	DATA_BLOCK DB163
	TITLE =DBG063M  AERATION AIR STEEPING 16
	//COPYRIGHT:    (C) 2009  BUHLER AG, CH-9240 UZWIL, SWITZERLAND
	//
	//PRODUCT:      WinCoS_BIW01_09
	//
	//TITLE:        AERATION AIR STEEPING 16
	//                Machine group DB
	//                Maschinengruppen-DB
	//
	//-------------------------------------------------------------------------
	//
	//IDENT:        AUTHOR:             DEPT:             DATE:
	//
	//P01_DB163.1.0 K.Renz              CSB41             13.Jan.2010
	//              1st Release
	//
	//-------------------------------------------------------------------------
	//
	//PURPOSE:
	//
	//MANUAL :
	//
	//RESTRICTIONS:
	//
	//-------------------------------------------------------------------------
	AUTHOR  : KR
	FAMILY  : USW
	NAME    : DBG063M
	VERSION : 00.00

	FB163
	BEGIN
	      #Gr.Par.ParObjectNo 	:=6300;
	      #Gr.Par.ParIdling      	:=2;
	      #Gr.Par.ParMgr	        :=True;
	      #Gr.Par.ParWgr	        :=False;
	      #Gr.Par.ParGgr	        :=False;
	      #Gr.Par.ParEmptyingTime 	:=0;
	      #Gr.Par.ParHornCode       :=1;
	//Parameter =A-1126-QXV/BZS41/42 : AERATION AIR RING ST 16
	      #A_1126_QXV_BZS41_42.Par.ParObjectNo                             :=6301;
	      #A_1126_QXV_BZS41_42.Par.ParMsgType                              :=7081;
	      #A_1126_QXV_BZS41_42.Par.ParHornCode                             :=1;
	      #A_1126_QXV_BZS41_42.Par.ParMonTime                              :=100;
	      #A_1126_QXV_BZS41_42.Par.ParPulseTimeHN                          :=5;
	      #A_1126_QXV_BZS41_42.Par.ParPulseTimeLN                          :=5;
	      #A_1126_QXV_BZS41_42.Par.ParIdlingTime                           :=0;
	      #A_1126_QXV_BZS41_42.Par.ParDelayTime                            :=0;
	      #A_1126_QXV_BZS41_42.Par.ParLogOff                               :=False;
	      #A_1126_QXV_BZS41_42.Par.ParManual                               :=True;
	      #A_1126_QXV_BZS41_42.Par.ParPulseValve                           :=False;
	      #A_1126_QXV_BZS41_42.Par.ParContValve                            :=True;
	      #A_1126_QXV_BZS41_42.Par.ParManualFlap                           :=False;
	//
	//
	END_DATA_BLOCK
